Omron CX-Programmer project NewProject (CX-Programmer 9.61)

# PLC NewPLC1: CP1H XA

## Global symbols (name address type ; comment)
0.00 BOOL  ; START
0.01 BOOL  ; STOP
0.02 BOOL  ; JOB_IN
0.03 BOOL  ; JOB_OUT
0.04 BOOL  ; DRILLUP
0.05 BOOL  ; POS_SEN
0.06 BOOL  ; DRILLDOWN
100.00 BOOL  ; M1
100.01 BOOL  ; M2
100.02 BOOL  ; M3
100.03 BOOL  ; M4
100.04 BOOL  ; M5
10.00 BOOL  ; CONVAYOR
10.01 BOOL  ; DRILL_DOWN_MOT
10.02 BOOL  ; DRILL_UP_MOT
T0001 BOOL  ; TIMER1
T0002 BOOL  ; TIMER2
T0003 BOOL  ; TIMER3

## Program NewProgram1 (cyclic task 0)

### Section Section1

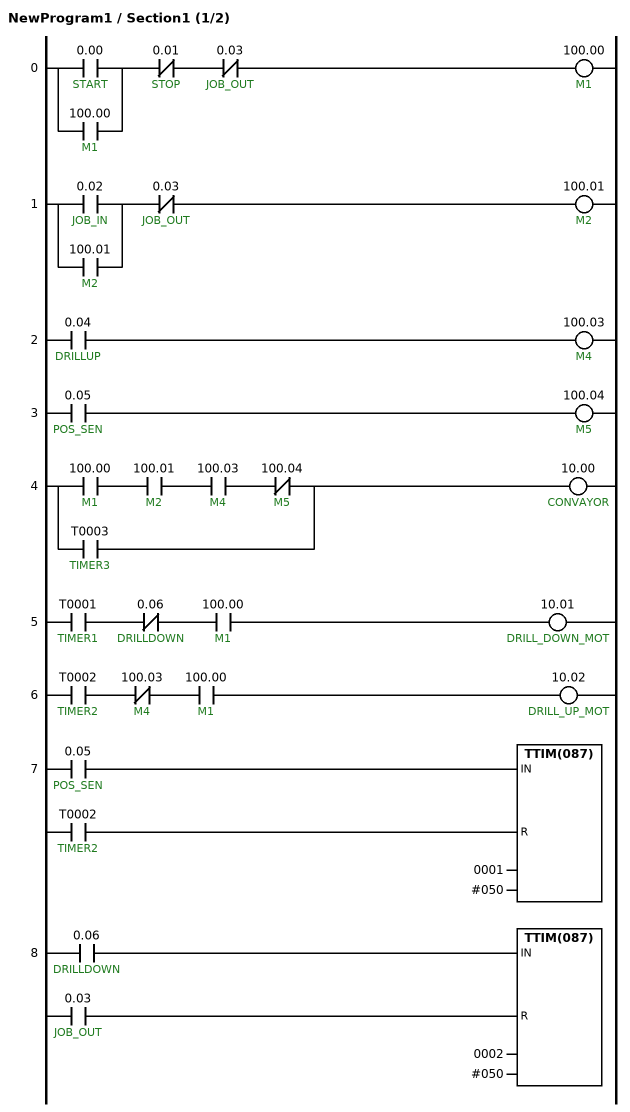
; rung 0
LD 0.00  ; START
OR 100.00  ; M1
ANDNOT 0.01  ; STOP
ANDNOT 0.03  ; JOB_OUT
OUT 100.00  ; M1
; rung 1
LD 0.02  ; JOB_IN
OR 100.01  ; M2
ANDNOT 0.03  ; JOB_OUT
OUT 100.01  ; M2
; rung 2
LD 0.04  ; DRILLUP
OUT 100.03  ; M4
; rung 3
LD 0.05  ; POS_SEN
OUT 100.04  ; M5
; rung 4
LD 100.00  ; M1
AND 100.01  ; M2
AND 100.03  ; M4
ANDNOT 100.04  ; M5
OR T0003  ; TIMER3
OUT 10.00  ; CONVAYOR
; rung 5
LD T0001  ; TIMER1
ANDNOT 0.06  ; DRILLDOWN
AND 100.00  ; M1
OUT 10.01  ; DRILL_DOWN_MOT
; rung 6
LD T0002  ; TIMER2
ANDNOT 100.03  ; M4
AND 100.00  ; M1
OUT 10.02  ; DRILL_UP_MOT
; rung 7
LD 0.05  ; POS_SEN
LD T0002  ; TIMER2
TTIM(087) 0001 #050  ; TIMER1
; rung 8
LD 0.06  ; DRILLDOWN
LD 0.03  ; JOB_OUT
TTIM(087) 0002 #050  ; TIMER2

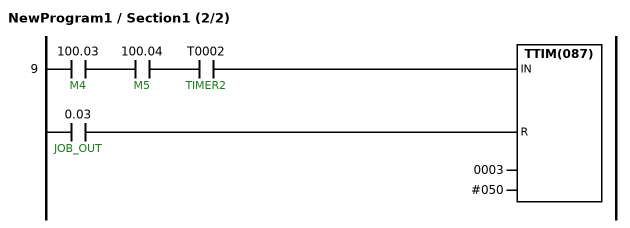
; rung 9
LD 100.03  ; M4
AND 100.04  ; M5
AND T0002  ; TIMER2
LD 0.03  ; JOB_OUT
TTIM(087) 0003 #050  ; TIMER3

### Section END
; rung 0
END(001)